TYPE ST_LaudaWriteCommands_Pump :
STRUCT
	Stage	: STRING := 'OUT_SP_01_';	// Pump stage 1-6 or 1-8 (device specific)
END_STRUCT
END_TYPE

(* stored: Version 1.1.0.1, ProductVersion 3.1.4024.12
   DUT ST_LaudaWriteCommands_Pump: Id {743ac91a-5542-4b70-b408-070137cbca3c} *)
